(* CoDeSys 2.3.9.41 project: Visual.pro *)
(* Libraries: Standard.lib 4.10.05 11:14:46, IecSfc.lib 13.4.06 15:51:28, SYSLIBCALLBACK.LIB 26.9.08 16:43:52 *)

(* Task configuration *)
TASK NewTask (PRIORITY := 1); (* freewheeling *)
	PLC_PRG();
	VIS_PRG();
END_TASK

(* Global variable list: Global_Variables *)
VAR_GLOBAL  (* 10 входов на 14 выходов *)
(* Входы *)
    (* Кнопки Push Buttons *)
	btnCallLevel1: BOOL;                  (* кнопка вызов кабины с 1 этажа         *)
	btnCallLevel2: BOOL;                  (*кнопка вызов кабины с 2 этажа              *)
	btnDownFromLevel1: BOOL;                (* Вниз с 1 этажа                          *)
	btnDownFromLevel2: BOOL;                 (* Вниз со 2 этажа                         *)
 btnUpOnLevel1: BOOL;                (* Вверх на 1 этаж                          *)
  btnUpOnLevel2: BOOL;                 (* Вверх на 2 этаж                         *)
	(* Кнопки-переключатели Switch Buttons *)
	SBEVlv:  BOOL; (* переключатель "Открыть аварийный клапан"       *)
    (* Датчики Sensors *)
	closedLevel1: BOOL;     (* датчик закрытых дверей  этаж 1         *)
	levelDetector: BOOL;     (* датчик этажа               *)
	closedLevel2: BOOL;     (* датчик закрытых дверей  этаж 2               *)
	closedLevel0: BOOL;     (*  датчик закрытых дверей  этаж 0                *)
(* Выходы *)
	(* Приводы/Лампы *)
	moveUpDetector: BOOL;    (* режим движения вверх                               *)
	moveDownDetector: BOOL;    (* режим движения вниз                             *)
	runEngine: BOOL;    (* запустить двигатель                       *)

	(* Команды/Лампы *)
       (* Этаж 0 *)
	closeDoorOnLevel0: BOOL;   (* дверь закрыта на этаже 0                               *)
	stopedOnLevel0: BOOL;   (* кабина стоит на этаже 0                               *)
	upOnLevel1: BOOL;   (* вверх на этаж 1                               *)
	upOnLevel2: BOOL;   (* вверх на этаж 2                               *)

      (* Этаж 1 *)
	closeDoorOnLevel1: BOOL;   (* дверь закрыта на этаже 1                               *)
	stopedOnLevel1: BOOL;   (* кабина стоит на этаже 1                               *)
	callOnLevel1: BOOL;   (* вызов на этаж 1                               *)
	down1OnLevel0: BOOL;   (* вниз на этаж 0                               *)

     (* Этаж 2 *)
	closeDoorOnLevel2: BOOL;   (* дверь закрыта на этаже 2                               *)
	stopedOnLevel2: BOOL;   (* кабина стоит на этаже 2                               *)
	callOnLevel2: BOOL;   (* вызов на этаж 2                               *)
	down2OnLevel0: BOOL;   (* вниз на этаж 0                               *)

	(* Лампы *)
	lelvel0: BOOL;
	lelvel1: BOOL;
	lelvel2: BOOL;
	engine: BOOL;

END_VAR

(* POU PLC_PRG, ST *)
PROGRAM PLC_PRG
VAR
	(*_TS1: BOOL;
	TS1: BOOL;
	_TS2: BOOL;
	TS2: BOOL;
	_MS: BOOL;
	MS: BOOL;
	_WTS: BOOL;
	WTS: BOOL;
	MtrTmr: BOOL;
	_Mtr: BOOL;
	WTSLmp: BOOL; *)
	level0: BOOL;
	level1: BOOL;
	level2: BOOL;
	callOnLevel2: BOOL;
END_VAR
(* ------- Состояния/Лампы ------- *)
(*
IF NOT _C1InMx AND     LS0 AND _Vlv1 AND _TS1 THEN C1InMx:=1;                    (* C1InMx+ *)
ELSIF  _C1InMx AND NOT LS0                    THEN C1InMx:=0;                    (* C1InMx- *)
END_IF;
IF NOT _C2InMx AND     LS0 AND _Vlv2 AND _TS2 THEN C2InMx:=1;                    (* C2InMx+ *)
ELSIF  _C2InMx AND NOT LS0                    THEN C2InMx:=0;                    (* C2InMx- *)
END_IF;
IF NOT _MxIsBd AND     LS0 AND _EVlv AND NOT _MxIsFn AND _C2InMx THEN MxIsBd:=1; (* MxIsBd+ *)
ELSIF  _MxIsBd AND NOT LS0                                       THEN MxIsBd:=0; (* MxIsBd- *)
END_IF;
IF NOT _MxIsFn AND     LS0 AND MtrTmr.Q AND NOT MxIsBd THEN MxIsFn:=1;           (* MxIsFn+ *)
ELSIF  _MxIsFn AND NOT LS0                             THEN MxIsFn:=0;           (* MxIsFn- *)
END_IF;
(* ------- Вспомогательные переменные ------- *)
Fin:= (PBCmpl OR _Compl) AND NOT _Vlv1 AND NOT LS0 OR HtrErr OR MtrErr OR MxIsBd OR SBEVlv OR PBStop
                                                   OR NOT TS1 AND NOT LS1 AND NOT MxIsFn
                                                   OR NOT TS2 AND NOT LS2 AND NOT MxIsFn;
(* ------- Состояния/Лампы ------- *)
IF NOT _SysOn AND PBStrt AND NOT Fin THEN SysOn:=1;                              (* SysOn+  *)
ELSIF  _SysOn AND                Fin THEN SysOn:=0;                              (* SysOn-  *)
END_IF;
IF NOT _Compl AND     SysOn AND PBCmpl THEN Compl:=1;                            (* Compl+  *)
ELSIF  _Compl AND NOT SysOn            THEN Compl:=0;                            (* Compl-  *)
END_IF;
(* ------- Приводы/Лампы ------- *)
EVlv:=SBEVlv;
Vlv1:=SysOn AND TS1 AND NOT LS1 AND NOT C2InMx AND NOT(Compl AND NOT LS0) AND WTS;
Vlv2:=SysOn AND TS2 AND     LS1 AND NOT LS2 AND NOT MxIsFn AND WTS;
Mtr :=SysOn AND LS2 AND NOT MxIsFn AND WTS AND C1InMx AND C2InMx;
PVlv:=SysOn AND             MxIsFn;
(* ------- Нагреватель/Лампа ------- *)
IF NOT _Htr AND      SysOn AND NOT LTS  THEN Htr:=1; (* Htr+ *)
ELSIF  _Htr AND (NOT SysOn OR      UTS) THEN Htr:=0; (* Htr- *)
END_IF;
(* ------- Лампы ------- *)
TS1Lmp:= NOT TS1;                                                                (* TS1Lmp  *)
TS2Lmp:= NOT TS2;                                                                (* TS2Lmp  *)
LS0Lmp:= LS0;                                                                    (* LS0Lmp  *)
LS1Lmp:= LS1;                                                                    (* LS1Lmp  *)
LS2Lmp:= LS2;                                                                    (* LS2Lmp  *)
MSLmp := MS;                                                                     (* MSLmp   *)
UTSLmp:= UTS;                                                                    (* UTSLmp  *)
LTSLmp:= LTS;                                                                    (* LTSLmp  *)
WTSLmp:= WTS;                                                                    (* WTSLmp  *)
*)

level0:= stopedOnLevel0 AND NOT runEngine;
level1:= stopedOnLevel1 AND NOT runEngine;
level2:= stopedOnLevel2 AND NOT runEngine;

upOnLevel1:= stopedOnLevel0 AND btnUpOnLevel1;
IF(NOT runEngine AND stopedOnLevel1)
THEN upOnLevel1:=FALSE;
END_IF;

upOnLevel2:= stopedOnLevel0 AND btnUpOnLevel2;
IF(NOT runEngine AND stopedOnLevel2)
THEN upOnLevel2:=FALSE;
END_IF;

callOnLevel1:=(btnCallLevel1 AND NOT stopedOnLevel1 AND NOT runEngine);
IF(stopedOnLevel1 AND NOT runEngine)
THEN callOnLevel1:=FALSE;
END_IF;

callOnLevel2:=(btnCallLevel2 AND NOT stopedOnLevel2 AND NOT runEngine);
IF(stopedOnLevel2 AND NOT runEngine)
THEN callOnLevel2:=FALSE;
END_IF;

down1OnLevel0:= NOT runEngine AND stopedOnLevel1 AND (btnDownFromLevel1 ); (* Проверку 10 секунд *)
IF(NOT runEngine AND stopedOnLevel0)
THEN down1OnLevel0:=FALSE;
END_IF;

down2OnLevel0:=NOT runEngine AND stopedOnLevel2 AND (btnDownFromLevel2); (*Условие времени добавить *)
IF NOT (runEngine AND stopedOnLevel0)
THEN down2OnLevel0:=FALSE;
END_IF;
(* ------- Псевдооператорный раздел ------- *)
(*_MtrErr:=MtrErr; _HtrErr:=HtrErr; _C1InMx:=C1InMx; _C2InMx:=C2InMx;  _MxIsFn:=MxIsFn; _MxIsBd:=MxIsBd;
_SysOn:=SysOn; _Compl:=Compl;
_EVlv:=EVlv; _Vlv1:=Vlv1; _Vlv2:=Vlv2; _Mtr:=Mtr; _Htr:=Htr;
_TS1:=TS1; _TS2:=TS2; _MS :=MS; _WTS:=WTS;
*)
(* ------- Лампа включенного двигателя ------- *)
runEngine:= closedLevel0 AND closedLevel1 AND closedLevel2 AND(NOT stopedOnLevel0 AND NOT stopedOnLevel1 AND NOT stopedOnLevel2 AND
							(upOnLevel1 OR upOnLevel2 OR down2OnLevel0 OR down1OnLevel0));
END_PROGRAM

(* POU VIS_PRG, ST *)
PROGRAM VIS_PRG
VAR
  (* ------- Обычные кнопки ------- *)
  callLevel1: BOOL;                  (*  вызов кабины с 1 этажа (синий)                *)
  callLevel2: BOOL;                  (* вызов кабины с 2 этажа (синий)             *)
  downFromLevel1: BOOL;                (* Вниз с 1 этажа                          *)
  downFromLevel2: BOOL;                 (* Вниз со 2 этажа                         *)
 upOnLevel1: BOOL;                (* Вверх на 1 этаж                          *)
  upOnLevel2: BOOL;                 (* Вверх на 2 этаж                         *)
  (* ------- Кнопки-переключатели ------- *)
  SBMtrBrk: BOOL;                (* поломка привода мешалки                *)
  SBHtrBrk: BOOL;                (* поломка нагревателя                    *)
  (* ------- Жидкости ------- *)
  Cmp1, _Cmp1: INT;              (* объем компонента 1 (синего)   в баке 1 *)
  Cmp2, _Cmp2: INT;              (* объем компонента 2 (красного) в баке 2 *)
  Mix,   _Mix: INT;              (* объем смеси в резервуаре               *)
  MixClr:      DWORD;            (* цвет  смеси в резервуаре               *)
  Red,   _Red: REAL;             (* коэффициент красного цвета в смеси     *)
  (* ------- Нагреватель ------- *)
  HtrClr: DWORD:=16#00_FF_FF_FF; (* температура нагревателя (цвет)         *)
  HtrRed, _HtrRed: BYTE;         (* степень накаливания нагревателя        *)
  HtrOn: BOOL;                   (* нагреватель функционирует (греет)      *)
	closedLevel1: BOOL;
	closedLevel2: BOOL;
	closedLevel0: BOOL;
	levelDetector: BOOL;
END_VAR
(* объем каждого из баков --- 300 единиц *)
(* пропускная способность каждого клапана равняется 1 единице за время прохода рабочего цикла ПЛК *)
(* но отрисовывать уменьшение объема жидкости в баке нужно в 3 раза медленне, чем происходит отрисовка заполнеия резервуара для смешивания *)
(* считается, что все клапаны обладают одинаковой пропускной способностью *)

(* Мы - рассчитываем по датчикам когда горят лампы *)
(* Cmp1:= MAX(0,MIN(360,BOOL_TO_INT(NOT PBCmp1)*_Cmp1+BOOL_TO_INT(PBTnk1)*360-BOOL_TO_INT(Vlv1)));
Cmp2:= MAX(0,MIN(240,BOOL_TO_INT(NOT PBCmp2)*_Cmp2+BOOL_TO_INT(PBTnk2)*240-BOOL_TO_INT(Vlv2)));
Mix := MAX(0,_Mix
             +BOOL_TO_INT(Vlv1 AND _Cmp1>0)
             +BOOL_TO_INT(Vlv2 AND _Cmp2>0)
             -BOOL_TO_INT(EVlv AND _Mix >0)
             -BOOL_TO_INT(PVlv AND _Mix >0)
          ); 
Red := BOOL_TO_INT(Mix>0)*(_Red*_Mix+1*BOOL_TO_INT(Vlv2 AND _Cmp2>0)
                                    -1*_Red*BOOL_TO_INT(PVlv AND _Mix >0)
                                    -1*_Red*BOOL_TO_INT(EVlv AND _Mix >0)
                                                                         )/MAX(1,Mix);
MixClr := 65536*REAL_TO_BYTE(255*(1-Red))+REAL_TO_BYTE(255*Red);
(* ------- Нагреватель ------- *)
HtrOn:=Htr AND NOT SBHtrBrk; (* нагреватель включается, если не сломан       *)
HtrRed:=_HtrRed+BOOL_TO_BYTE(HtrOn AND _HtrRed<255)-BOOL_TO_BYTE(NOT HtrOn AND _HtrRed>0);
HtrClr:=65536*(255-HtrRed)+256*(255-HtrRed)+255;
(* ------- Выставление сигналов датчиков ------- *)


levelDetector:=((moveUpDetector==FALSE) && (moveDownDetector==FALSE) );             (* датчик этажа *)                 *)
(* -------  Псевдооператорный раздел ------- *)
(*  _Cmp1:=Cmp1; _Cmp2:=Cmp2; _Mix:=Mix; _Red:=Red; _HtrRed:=HtrRed;
*)
(*Закрыты ли все двери*)
closedLevel1:=(Cmp1>0);               (* датчик закрытых дверей  этаж 1        *)
closedLevel2:=(Cmp1>0);               (* датчик закрытых дверей  этаж 2        *)
closedLevel0:=(Cmp1>0);               (* датчик закрытых дверей  этаж 0        *)
END_PROGRAM

(* Visualisation Vis
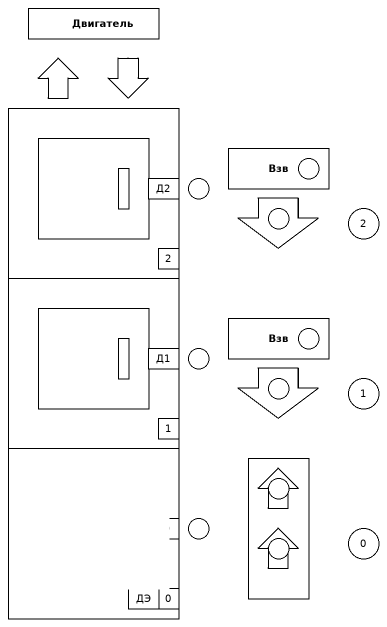
rectangle at (380,160)-(481,201): text "Взв"; shows .MtrTmr.ET
ellipse at (450,170)-(471,191): taps .callLevel2
ellipse at (500,220)-(531,251): text "2"
ellipse at (500,390)-(531,421): text "1"
ellipse at (500,540)-(531,571): text "0"
rectangle at (300,190)-(331,211): text "Д2"
rectangle at (310,260)-(331,281): text "2"
rectangle at (300,360)-(331,381): text "Д1"
rectangle at (310,430)-(331,451): text "1"
rectangle at (300,530)-(331,551): text "Д0"
rectangle at (310,600)-(331,621): text "0"
ellipse at (420,220)-(441,241): taps .downFromLevel2
rectangle at (380,330)-(481,371): text "Взв"; shows .MtrTmr.ET
ellipse at (450,340)-(471,361): taps .callLevel1
ellipse at (420,390)-(441,411): taps .downFromLevel1
rectangle at (280,600)-(311,621): text "ДЭ"
ellipse at (420,490)-(441,511): taps .callLevel2
ellipse at (420,550)-(441,571): taps .callLevel1
rectangle at (180,20)-(311,51): text "Двигатель"
20 more shapes without text or variables
*)
